TYPE BoxesCom :
STRUCT
  IndexOfFirst : DINT;
  IndexOfNext : DINT;
  Buffer : ARRAY [0..20] OF Box;
END_STRUCT
END_TYPE

(* stored: Version 1.1.0.1
   DUT BoxesCom: Id {08fe2898-bba2-4e9c-876d-d6b5306c5b83} *)
